PROGRAM PRG_03_VibrationAnalytics
VAR
	VibSensor					: ARRAY [1..6] OF VibrationSensor;
	
	
	{attribute 'OPC.UA.DA' := '0'}
	{attribute 'OPC.UA.DA.Access' := '1'}			// read only
	{attribute 'OPC.UA.DA.StructuredType' := '1'}
	VibSensorStruct01			: VibAccelarationDataModel;
	
	{attribute 'OPC.UA.DA' := '0'}
	{attribute 'OPC.UA.DA.Access' := '1'}			// read only
	{attribute 'OPC.UA.DA.StructuredType' := '1'}
	VibSensorStruct02			: VibAccelarationDataModel;

	{attribute 'OPC.UA.DA' := '0'}
	{attribute 'OPC.UA.DA.Access' := '1'}			// read only
	{attribute 'OPC.UA.DA.StructuredType' := '1'}
	VibSensorStruct03			: VibAccelarationDataModel;
	
	{attribute 'OPC.UA.DA' := '0'}
	{attribute 'OPC.UA.DA.Access' := '1'}			// read only
	{attribute 'OPC.UA.DA.StructuredType' := '1'}
	VibSensorStruct04			: VibAccelarationDataModel;
	
	{attribute 'OPC.UA.DA' := '0'}
	{attribute 'OPC.UA.DA.Access' := '1'}			// read only
	{attribute 'OPC.UA.DA.StructuredType' := '1'}
	VibSensorStruct05			: VibAccelarationDataModel;
	
	{attribute 'OPC.UA.DA' := '0'}
	{attribute 'OPC.UA.DA.Access' := '1'}			// read only
	{attribute 'OPC.UA.DA.StructuredType' := '1'}
	VibSensorStruct06			: VibAccelarationDataModel;
	

END_VAR


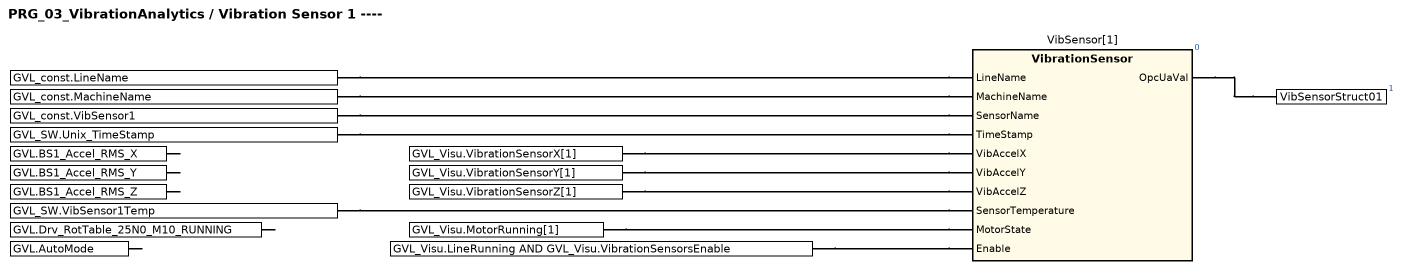
// PAGE Vibration Sensor 1 ----
VibSensor[1](
    LineName := GVL_const.LineName,
    MachineName := GVL_const.MachineName,
    SensorName := GVL_const.VibSensor1,
    TimeStamp := GVL_SW.Unix_TimeStamp,
    VibAccelX := GVL_Visu.VibrationSensorX[1],
    VibAccelY := GVL_Visu.VibrationSensorY[1],
    VibAccelZ := GVL_Visu.VibrationSensorZ[1],
    SensorTemperature := GVL_SW.VibSensor1Temp,
    MotorState := GVL_Visu.MotorRunning[1],
    Enable := GVL_Visu.LineRunning AND GVL_Visu.VibrationSensorsEnable); // VibrationSensor
VibSensorStruct01 := VibSensor[1].OpcUaVal;

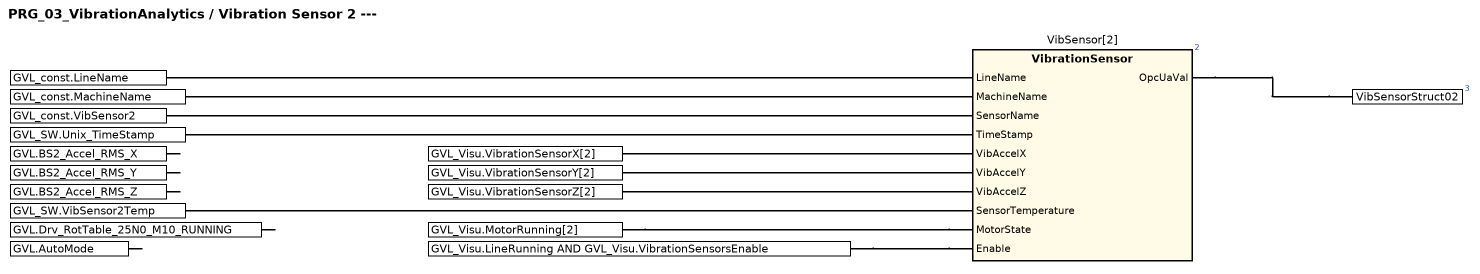
// PAGE Vibration Sensor 2 ---
VibSensor[2](
    LineName := GVL_const.LineName,
    MachineName := GVL_const.MachineName,
    SensorName := GVL_const.VibSensor2,
    TimeStamp := GVL_SW.Unix_TimeStamp,
    VibAccelX := GVL_Visu.VibrationSensorX[2],
    VibAccelY := GVL_Visu.VibrationSensorY[2],
    VibAccelZ := GVL_Visu.VibrationSensorZ[2],
    SensorTemperature := GVL_SW.VibSensor2Temp,
    MotorState := GVL_Visu.MotorRunning[2],
    Enable := GVL_Visu.LineRunning AND GVL_Visu.VibrationSensorsEnable); // VibrationSensor
VibSensorStruct02 := VibSensor[2].OpcUaVal;

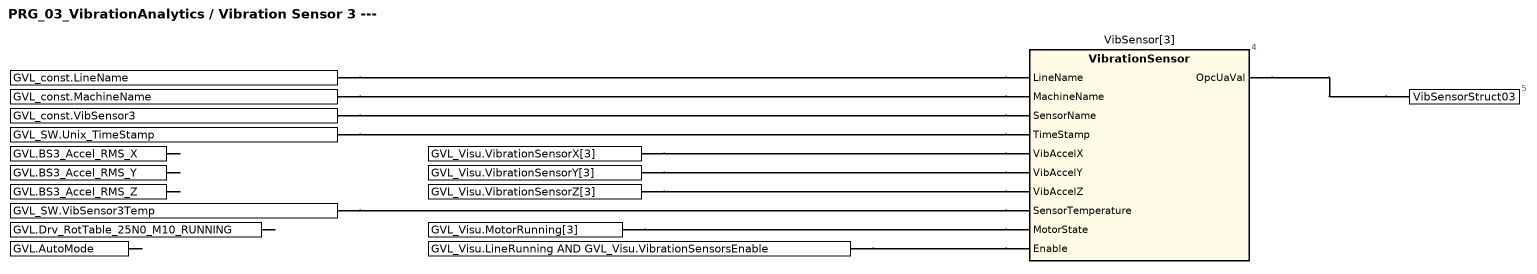
// PAGE Vibration Sensor 3 ---
VibSensor[3](
    LineName := GVL_const.LineName,
    MachineName := GVL_const.MachineName,
    SensorName := GVL_const.VibSensor3,
    TimeStamp := GVL_SW.Unix_TimeStamp,
    VibAccelX := GVL_Visu.VibrationSensorX[3],
    VibAccelY := GVL_Visu.VibrationSensorY[3],
    VibAccelZ := GVL_Visu.VibrationSensorZ[3],
    SensorTemperature := GVL_SW.VibSensor3Temp,
    MotorState := GVL_Visu.MotorRunning[3],
    Enable := GVL_Visu.LineRunning AND GVL_Visu.VibrationSensorsEnable); // VibrationSensor
VibSensorStruct03 := VibSensor[3].OpcUaVal;

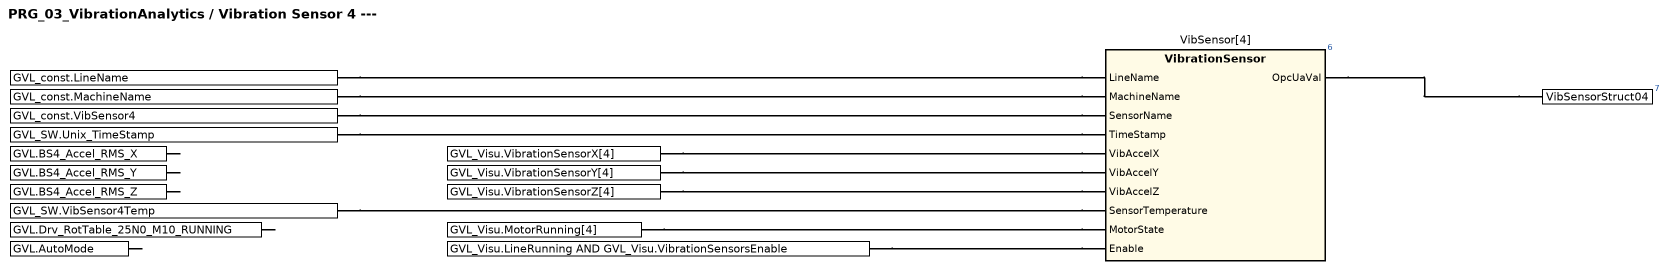
// PAGE Vibration Sensor 4 ---
VibSensor[4](
    LineName := GVL_const.LineName,
    MachineName := GVL_const.MachineName,
    SensorName := GVL_const.VibSensor4,
    TimeStamp := GVL_SW.Unix_TimeStamp,
    VibAccelX := GVL_Visu.VibrationSensorX[4],
    VibAccelY := GVL_Visu.VibrationSensorY[4],
    VibAccelZ := GVL_Visu.VibrationSensorZ[4],
    SensorTemperature := GVL_SW.VibSensor4Temp,
    MotorState := GVL_Visu.MotorRunning[4],
    Enable := GVL_Visu.LineRunning AND GVL_Visu.VibrationSensorsEnable); // VibrationSensor
VibSensorStruct04 := VibSensor[4].OpcUaVal;

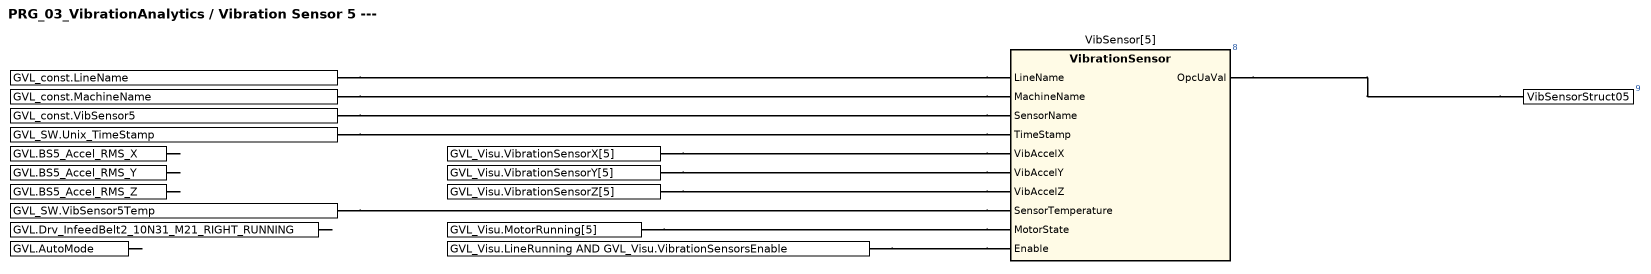
// PAGE Vibration Sensor 5 ---
VibSensor[5](
    LineName := GVL_const.LineName,
    MachineName := GVL_const.MachineName,
    SensorName := GVL_const.VibSensor5,
    TimeStamp := GVL_SW.Unix_TimeStamp,
    VibAccelX := GVL_Visu.VibrationSensorX[5],
    VibAccelY := GVL_Visu.VibrationSensorY[5],
    VibAccelZ := GVL_Visu.VibrationSensorZ[5],
    SensorTemperature := GVL_SW.VibSensor5Temp,
    MotorState := GVL_Visu.MotorRunning[5],
    Enable := GVL_Visu.LineRunning AND GVL_Visu.VibrationSensorsEnable); // VibrationSensor
VibSensorStruct05 := VibSensor[5].OpcUaVal;

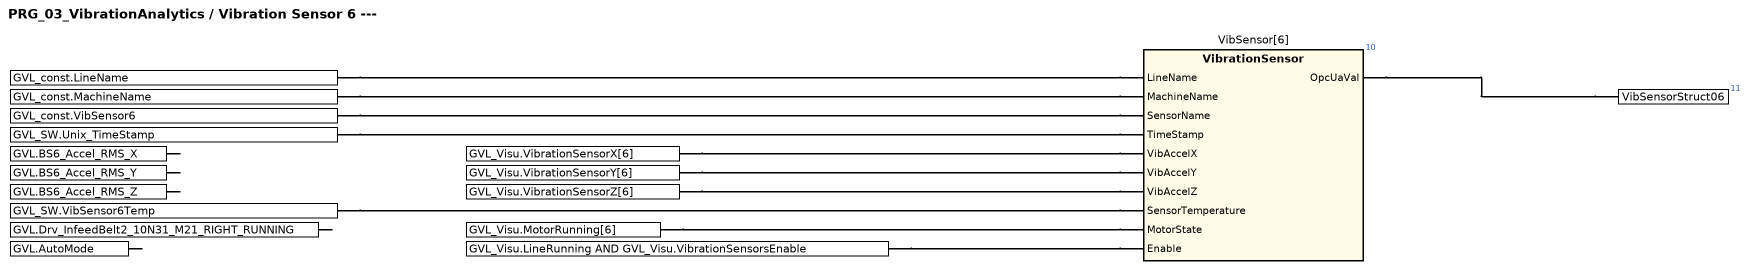
// PAGE Vibration Sensor 6 ---
VibSensor[6](
    LineName := GVL_const.LineName,
    MachineName := GVL_const.MachineName,
    SensorName := GVL_const.VibSensor6,
    TimeStamp := GVL_SW.Unix_TimeStamp,
    VibAccelX := GVL_Visu.VibrationSensorX[6],
    VibAccelY := GVL_Visu.VibrationSensorY[6],
    VibAccelZ := GVL_Visu.VibrationSensorZ[6],
    SensorTemperature := GVL_SW.VibSensor6Temp,
    MotorState := GVL_Visu.MotorRunning[6],
    Enable := GVL_Visu.LineRunning AND GVL_Visu.VibrationSensorsEnable); // VibrationSensor
VibSensorStruct06 := VibSensor[6].OpcUaVal;
// GVL.BS1_Accel_RMS_X: input not connected
// GVL.BS1_Accel_RMS_Y: input not connected
// GVL.BS1_Accel_RMS_Z: input not connected
// GVL.Drv_RotTable_25N0_M10_RUNNING: input not connected
// GVL.AutoMode: input not connected
// GVL.BS2_Accel_RMS_X: input not connected
// GVL.BS2_Accel_RMS_Y: input not connected
// GVL.BS2_Accel_RMS_Z: input not connected
// GVL.Drv_RotTable_25N0_M10_RUNNING: input not connected
// GVL.AutoMode: input not connected
// GVL.BS3_Accel_RMS_X: input not connected
// GVL.BS3_Accel_RMS_Y: input not connected
// GVL.BS3_Accel_RMS_Z: input not connected
// GVL.Drv_RotTable_25N0_M10_RUNNING: input not connected
// GVL.AutoMode: input not connected
// GVL.BS4_Accel_RMS_X: input not connected
// GVL.BS4_Accel_RMS_Y: input not connected
// GVL.BS4_Accel_RMS_Z: input not connected
// GVL.Drv_RotTable_25N0_M10_RUNNING: input not connected
// GVL.AutoMode: input not connected
// GVL.BS5_Accel_RMS_X: input not connected
// GVL.BS5_Accel_RMS_Y: input not connected
// GVL.BS5_Accel_RMS_Z: input not connected
// GVL.Drv_InfeedBelt2_10N31_M21_RIGHT_RUNNING: input not connected
// GVL.AutoMode: input not connected
// GVL.BS6_Accel_RMS_X: input not connected
// GVL.BS6_Accel_RMS_Y: input not connected
// GVL.BS6_Accel_RMS_Z: input not connected
// GVL.Drv_InfeedBelt2_10N31_M21_RIGHT_RUNNING: input not connected
// GVL.AutoMode: input not connected

END_PROGRAM

(* stored: Version 1.1.0.1, ProductVersion 3.1.4024.15
   POU PRG_03_VibrationAnalytics: Id {df3a27d8-7441-46ff-a708-961eecefb8af}, SpecialFunc None *)
